Staubli VAL3: onEnterEvent.pgx

program onEnterEvent(tool& x_tTool[])
begin
  //
  // NB sEvent is the selected
  // element in the LIST
  //
  call editTool(x_tTool)
  call tcp:setTool(x_tTool,nIndexTool)
  logMsg("[KERNEL] INTERFACE:Change value of the tool :"+toString("",nIndexTool))
  //
end
